{attribute 'GeneratedUsingTerminal: KL6771-0002'}
{attribute addProperty BoxType "KL6771-0002"}
{attribute addProperty Id "Channel_1AT %Q*Channel_6931CC5B0"}
{attribute addProperty CRC "1384833944"}
{attribute addProperty Size "0"}
TYPE KL_528AE398 :
STRUCT
	{attribute addProperty Name "Channel_1"}
	Channel_1 : Channel_6931CC5B;
END_STRUCT
END_TYPE

(* stored: Version 1.2.0.0, ProductVersion 3.1.4024.9
   DUT KL_528AE398: Id {d783836a-1dc2-48ca-9f83-d0832fc00ec9} *)
